# EPICS autosave request: autosave/galil_analog_in.req
$(P)$(R)Deadb_SP
